{attribute 'qualified_only'}
VAR_GLOBAL CONSTANT
END_VAR

(* stored: Version 1.1.0.1, ProductVersion 3.1.4024.12
   GVL Param: Id {7502923b-646d-49fa-b13a-71e80a630643}, ParameterList True *)
